FUNCTION_BLOCK FB_AnalogDeviceRampControl
VAR
	i : INT;
END_VAR

FOR i:=1 TO E_aAnalogInputIO_Index.E_PV_EPC_04 DO
	GVL_IO.aAnalogOutputIO[i] := LREAL_TO_INT(GVL_IO.aAnalogController[i].cvController.rControlValue / GVL_CONSTANT.AnalogControllerOutputVoltage * GVL_CONSTANT.EL3064MaxValueH); //Write to Device
	GVL_IO.aAnalogController[i].cvController();
END_FOR


//jhkang aController 의 Input은 언제 들어감?
//Temp Controller
GVL_IO.wE3508_CV := LREAL_TO_WORD(GVL_IO.aAnalogController[E_aAnalogInputIO_Index.E_PV_Susceptor_Temp].cvController.rControlValue * 10 )  ; //Write to Temperature Controller
GVL_IO.aAnalogController[E_aAnalogInputIO_Index.E_PV_Susceptor_Temp].cvController();

//Temp Pressure Controller				
GVL_IO.wIqPlus_CV := LREAL_TO_WORD(GVL_IO.aAnalogController[E_aAnalogInputIO_Index.E_PV_Reactor_Pressure].cvController.rControlValue); //Write to Pressure Controller
GVL_IO.aAnalogController[E_aAnalogInputIO_Index.E_PV_Reactor_Pressure].cvController();

//Rotation Controller		
GVL_IO.rRotation_ControlValue := LREAL_TO_REAL(GVL_IO.aAnalogController[E_aAnalogInputIO_Index.E_PV_susceptorRotation].cvController.rControlValue); //Write to Rotation Controller (rpm)
GVL_IO.aAnalogController[E_aAnalogInputIO_Index.E_PV_susceptorRotation].cvController();

END_FUNCTION_BLOCK

(* stored: Version 1.1.0.1, ProductVersion 3.1.4026.11
   POU FB_AnalogDeviceRampControl: Id {901ef948-d319-4e50-9c34-c06b07342954}, SpecialFunc None *)
